FUNCTION_BLOCK CL_AxisDriverL2RightFront EXTENDS CL_AxisDriverAX8206
VAR
END_VAR

SUPER^();

METHOD PUBLIC Init : BOOL
VAR_INPUT  
  stDriver : POINTER TO ST_DriverAX8206_HWI;
END_VAR
Init := FALSE;
IF stDriver <> 0 THEN
  Init := SUPER^.InitDriver(stDriverCom_P := ADR(stDriver^.comState), stDriverCh_P := ADR(stDriver^.stFront));
END_IF
END_METHOD

METHOD PROTECTED InitDefect : BOOL
VAR_INPUT
END_VAR
InitDefect := SUPER^.InitDefect();
ADSLOGSTR(ADSLOG_MSGTYPE_LOG, 'CL_AxisDriverL2RightFront init defect','');
END_METHOD

END_FUNCTION_BLOCK

(* stored: Version 1.1.0.1, ProductVersion 3.1.4024.12
   POU CL_AxisDriverL2RightFront: Id {86cba96c-6c59-47e7-878d-6c1ffbc0e78e}, SpecialFunc None
   Method Init: Id {814b90a8-7739-4e64-bc14-5598323eb8e5}
   Method InitDefect: Id {0c2e11c5-a079-451a-9d62-a795ed63e243} *)
